PROGRAM MAIN
VAR
	bInit				: BOOL;	

	fMotorCurrent		AT %I* : LREAL;
	fTemperature		AT %I* : LREAL;
	fVibration			AT %I* : LREAL;
	nCycleTime			AT %I* : DINT;
	bCycleRun			AT %I* : BOOL;
	
	// user vars
	current_arr			: ARRAY[0..24] OF LREAL;
	vib_arr				: ARRAY[0..24] OF LREAL;
	
	fbStatsCurrent		: FB_ALY_ArrayStatistics;
	fbStatsVibration	: FB_ALY_ArrayStatistics;
	
	stFeatures			: ST_Features;
	
	i					: DINT;
	rtStart				: R_TRIG;
	ftEnd				: F_TRIG;
	
	bEnableLogging		: BOOL := FALSE;
	sFilePath			: STRING := 'C:\Temp\csv\test.csv';
	fbFile				: FB_FileIO;
	sData				: STRING(512);
	bWrite				: BOOL;
END_VAR

IF NOT bInit THEN
	fbStatsCurrent.Configure(FALSE, 0.1, 0.1, 0);
	fbStatsVibration.Configure(FALSE, 0.1, 0.1, 0);
	bInit := FALSE;
END_IF

rtStart(CLK:=bCycleRun);
ftEnd(CLK:=bCycleRun);

// reset
IF rtStart.Q THEN
	i := 0;
	MEMSET(ADR(current_arr[0]), 0, SIZEOF(LREAL) * 25);
	MEMSET(ADR(vib_arr[0]), 0, SIZEOF(LREAL) * 25);
	IF bEnableLogging THEN
		bWrite := TRUE;
	END_IF
END_IF

IF bCycleRun THEN
	IF i < 25 THEN
		current_arr[i] := fMotorCurrent;
		vib_arr[i] := fVibration;
	END_IF
	stFeatures.temp := fTemperature;
	stFeatures.cycle_time := nCycleTime;
	i := i + 1;
ELSE
	fbStatsCurrent.Call(ADR(current_arr), SIZEOF(current_arr));
	fbStatsVibration.Call(ADR(vib_arr), SIZEOF(vib_arr));
	
	IF fbStatsCurrent.bNewResult THEN
		stFeatures.curr_mean := fbStatsCurrent.fMean;
		stFeatures.curr_peak := fbStatsCurrent.fMax;
		stFeatures.curr_range := fbStatsCurrent.fMax - fbStatsCurrent.fMin;
		stFeatures.curr_delta_max := fbStatsCurrent.fMaxDelta;
		stFeatures.curr_delta_idx := fbStatsCurrent.nIdxMaxDelta;
		stFeatures.curr_std := fbStatsCurrent.fStandardDeviation;
	END_IF
	IF fbStatsVibration.bNewResult THEN
		stFeatures.vibe_mean := fbStatsVibration.fMean;
		stFeatures.vibe_peak := fbStatsVibration.fMax;
		stFeatures.vibe_range := fbStatsVibration.fMax - fbStatsVibration.fMin;
		stFeatures.vibe_delta_max := fbStatsVibration.fMaxDelta;
		stFeatures.vibe_delta_idx := fbStatsVibration.nIdxMaxDelta;
		stFeatures.vibe_std := fbStatsVibration.fStandardDeviation;
	END_IF
	
	IF fbStatsCurrent.bNewResult AND fbStatsVibration.bNewResult THEN
		sData := F_Feature_Csv(stFeatures);
	END_IF
END_IF

IF bWrite AND_THEN fbFile.AppendText(sFilePath, sData) THEN
	bWrite := FALSE;
END_IF

END_PROGRAM

(* stored: Version 1.1.0.1, ProductVersion 3.1.4026.18
   POU MAIN: Id {1dcddbdf-2253-4ac8-963c-afea778d61ce}, SpecialFunc None *)
